{attribute 'linkalways'} 
{attribute 'no_explicit_call' := 'This FB is a CLASS and must be accessed using methods or properties'}
{attribute 'enable_dynamic_creation'}
FUNCTION_BLOCK _ETcVnAdaptiveThresholdMethod EXTENDS EnumDatatypeBase
VAR
	localData : ETcVnAdaptiveThresholdMethod;
	activeData : REFERENCE TO ETcVnAdaptiveThresholdMethod;
	enumBaseDatatype : _DINT(localData);
END_VAR

METHOD PRIVATE AddLocalEnumeration
VAR_INPUT
	Enumeration : T_MAXSTRING;
	Value : ETcVnAdaptiveThresholdMethod;
END_VAR
AddEnumeration(Enumeration, Value);
END_METHOD

PROPERTY PUBLIC Address : PVOID
GET
Address := ADR(activeData);
END_GET
END_PROPERTY

METHOD PUBLIC ClearReference
VAR_INPUT
END_VAR
activeData REF= localData;
SetBaseDatatypeReference();
END_METHOD

METHOD PUBLIC Clone : I_Datatype
VAR
    pClone : POINTER TO _ETcVnAdaptiveThresholdMethod;
END_VAR
pClone := __NEW(_ETcVnAdaptiveThresholdMethod(InitialValue := Value));
Clone := pClone^;
END_METHOD

METHOD FB_init : BOOL
VAR_INPUT
	bInitRetains : BOOL; // if TRUE, the retain variables are initialized (warm start / cold start)
	bInCopyCode : BOOL;  // if TRUE, the instance afterwards gets moved into the copy code (online change)
	InitialValue : ETcVnAdaptiveThresholdMethod;
END_VAR
localData := InitialValue;
AddBaseDatatype(enumBaseDatatype);
ClearReference();

AddLocalEnumeration('TCVN_ATM_MEAN', ETcVnAdaptiveThresholdMethod.TCVN_ATM_MEAN);
AddLocalEnumeration('TCVN_ATM_GAUSSIAN', ETcVnAdaptiveThresholdMethod.TCVN_ATM_GAUSSIAN);
END_METHOD

PROPERTY PUBLIC Identifier : T_MAXSTRING
GET
Identifier := 'ETcVnAdaptiveThresholdMethod';
END_GET
END_PROPERTY

METHOD IsEnumeratorValueEqual : BOOL
VAR_INPUT
	Enumerator : I_KeyValueForwardEnumerator;
END_VAR
VAR
	storedValue : ETcVnAdaptiveThresholdMethod;
END_VAR
IF NOT Enumerator.TryGet(storedValue) THEN
	RETURN;
END_IF

IsEnumeratorValueEqual := storedValue = activeData;
END_METHOD

METHOD PUBLIC MakeReferenceTo
VAR_INPUT
	ReferenceTarget : REFERENCE TO ETcVnAdaptiveThresholdMethod;
END_VAR
activeData REF= ReferenceTarget;
SetBaseDatatypeReference();
END_METHOD

METHOD PROTECTED SetBaseDatatypeReference
VAR_INPUT
END_VAR
enumBaseDatatype.MakeReferenceTo(activeData);
END_METHOD

PROPERTY PUBLIC Size : UDINT
GET
Size := SIZEOF(activeData);
END_GET
END_PROPERTY

METHOD TryMakeReferenceTo : BOOL
VAR_INPUT
	Target : I_Datatype;
END_VAR
VAR
	pTargetData : POINTER TO ETcVnAdaptiveThresholdMethod;
END_VAR
IF NOT IsEquivalentTo(Target) THEN
	RETURN;
END_IF

pTargetData := Target.Address;
activeData REF= pTargetData^;
SetBaseDatatypeReference();
TryMakeReferenceTo := TRUE;
END_METHOD

PROPERTY PUBLIC Value : ETcVnAdaptiveThresholdMethod
GET
Value := activeData;
END_GET
SET
activeData := Value;
END_SET
END_PROPERTY

END_FUNCTION_BLOCK

(* stored: Version 1.1.0.1, ProductVersion 3.1.4024.13
   POU _ETcVnAdaptiveThresholdMethod: Id {9da01fc5-1dc4-4a4e-9352-a879d3ae8a31}, SpecialFunc None
   Folder Core: Id {1a0e7959-c568-0b1f-2adf-6519dd143395}
   Folder Protected: Id {1b9e1262-1a18-0b84-0ff7-65a7d9d7a08b}
   Folder Customize: Id {67a44fdd-2de1-0dc5-2c16-60cc26053cbe}
   Folder Constructor: Id {7af4fc30-79ac-48d7-8c10-05eac5cab723}
   Folder Private: Id {6ccc4ec8-13a7-416e-8470-14c877cb4dd6}
   Folder Protected: Id {0ddb8528-3074-48ca-9958-48b0bea28d12}
   Method AddLocalEnumeration: Id {3ca3e93c-18fd-4189-98e4-31dac1cef591}
   Property Address: Id {809dbf93-3ede-08c6-0a76-bea9bff7c2ad}
   Get Get: Id {605ac528-e5a1-064c-20af-aa4235e29bc3}
   Method ClearReference: Id {db545cb3-3b6e-0454-242b-738816091f45}
   Method Clone: Id {2e0ff545-a58c-4917-9c55-2dd8ed5a1471}
   Method FB_init: Id {545b9c1e-b947-40b7-b132-9779fe73e6a1}
   Property Identifier: Id {59628a3e-3174-4eac-8bb3-46de9c8e8706}
   Get Get: Id {fd939138-ad23-43ed-8194-b4ab2ee31a4b}
   Method IsEnumeratorValueEqual: Id {51ff6e63-d275-4e3c-8281-d1d197322afe}
   Method MakeReferenceTo: Id {3433abe8-9ea3-49d7-b377-346522fa6ca0}
   Method SetBaseDatatypeReference: Id {1c77742b-d22f-0981-2d01-d722de1cfcdd}
   Property Size: Id {b689c4b5-32c4-065c-0fa0-04b90edae93a}
   Get Get: Id {647a8c92-ece6-087a-1dc6-94f2143d8f0c}
   Method TryMakeReferenceTo: Id {d2a455c2-7f84-4807-a11a-b08020f5928a}
   Property Value: Id {87cc2e0c-d6cd-4d45-a674-e2d8a6a3aae2}
   Get Get: Id {00cd73ec-b809-4411-81cb-115f8a9570e3}
   Set Set: Id {5679032f-6f0f-4cc8-9e86-909a6187f413} *)
